// TIA Portal V20 export
FUNCTION_BLOCK "LAF_ManageAlarms"   // FB82, LAD
TITLE = LAF_ManageAlarms
AUTHOR : Siemens Digital Industries
FAMILY : LAF
// Mapping the ProDiag categories to the commands of the ModeStateManager.
// stored: Access Published, IsIECCheckEnabled true, MemoryReserve 100, SetENOAutomatically true
   VAR_INPUT
      proDiagState : SV_FB_State_V2;
   END_VAR
   VAR_OUTPUT
      parentAlarmDB : "LAF_typeAlarms";
      alarmDB : "LAF_typeAlarms";
      hmiInterfaceDB : "LAF_typeAlarms";
   END_VAR
   VAR_IN_OUT
      feedback : "LUC_typeEmFeedback";
   END_VAR
   VAR_TEMP
      temp : Bool;
   END_VAR
   VAR CONSTANT
      REPLACE : Bool;   // OEM: replace with ProDiag statuses that command unit state
   END_VAR
BEGIN

REGION Network 1: BLOCK INFO HEADER
   // SIEMENS AG / (c)Copyright 2024
   // ------------------------------------------------------------------------------
   // Title:            LAF_ManageAlarms
   // Comment/Function: Mapping the ProDiag categories to the commands of the ModeStateManager.
   // Library/Family:   Library of Automation Framework
   // Author:           Siemens Digital Industry
   // Tested with:      ---
   // Engineering:      TIA Portal V19
   // Restrictions:     -
   // Requirements:     ---
   // ------------------------------------------------------------------------------
   // Change log table:
   // Version  | Date       | Expert in charge       | Changes applied
   // ---------|------------|------------------------|------------------------------
   // 01.01.00 | 21.06.2024 | SIMATIC Systems Support
   //                         First released version
END_REGION

REGION Network 2: Stop command
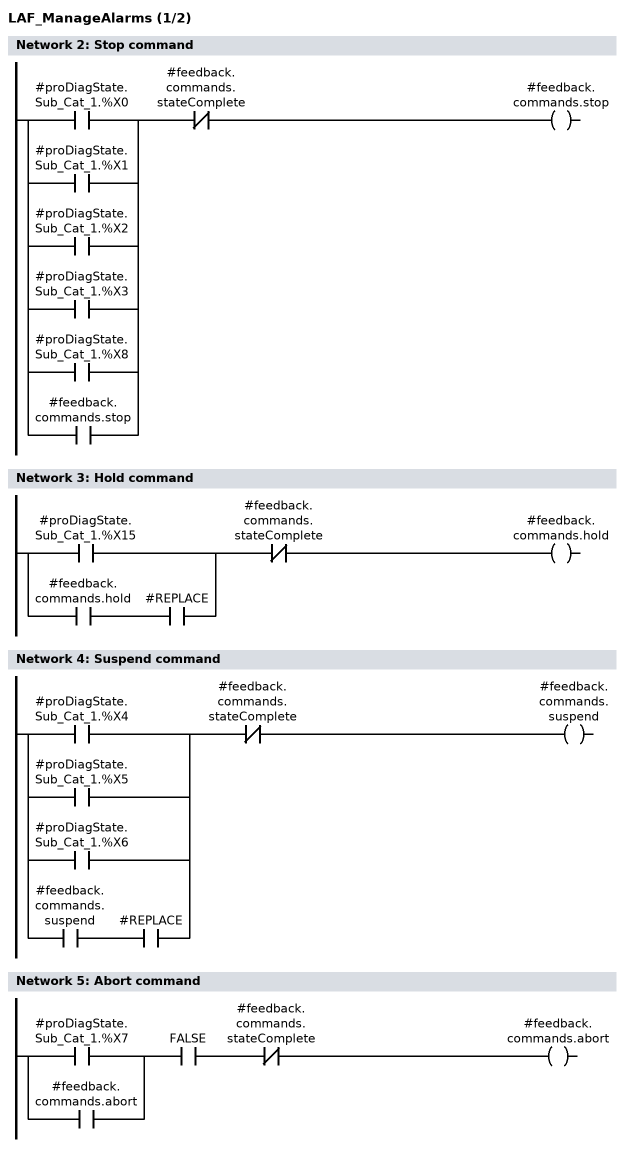
   RUNG wire#powerrail
      Contact( #proDiagState.Sub_Cat_1.%X0 )
      wire#w1
      I_Contact( #feedback.commands.stateComplete )
      Coil( #feedback.commands.stop )
   END_RUNG
   RUNG wire#powerrail
      Contact( #proDiagState.Sub_Cat_1.%X1 )
   END_RUNG wire#w1
   RUNG wire#powerrail
      Contact( #proDiagState.Sub_Cat_1.%X2 )
   END_RUNG wire#w1
   RUNG wire#powerrail
      Contact( #proDiagState.Sub_Cat_1.%X3 )
   END_RUNG wire#w1
   RUNG wire#powerrail
      Contact( #proDiagState.Sub_Cat_1.%X8 )
   END_RUNG wire#w1
   RUNG wire#powerrail
      Contact( #feedback.commands.stop )
   END_RUNG wire#w1
   // the same network as SCL:
   #feedback.commands.stop := (#proDiagState.Sub_Cat_1.%X0 OR #proDiagState.Sub_Cat_1.%X1 OR #proDiagState.Sub_Cat_1.%X2 OR #proDiagState.Sub_Cat_1.%X3 OR #proDiagState.Sub_Cat_1.%X8 OR #feedback.commands.stop) AND NOT #feedback.commands.stateComplete;
END_REGION

REGION Network 3: Hold command
   RUNG wire#powerrail
      Contact( #proDiagState.Sub_Cat_1.%X15 )
      wire#w1
      I_Contact( #feedback.commands.stateComplete )
      Coil( #feedback.commands.hold )
   END_RUNG
   RUNG wire#powerrail
      Contact( #feedback.commands.hold )
      Contact( #REPLACE )
   END_RUNG wire#w1
   // the same network as SCL:
   #feedback.commands.hold := (#proDiagState.Sub_Cat_1.%X15 OR (#feedback.commands.hold AND #REPLACE)) AND NOT #feedback.commands.stateComplete;
END_REGION

REGION Network 4: Suspend command
   RUNG wire#powerrail
      Contact( #proDiagState.Sub_Cat_1.%X4 )
      wire#w1
      I_Contact( #feedback.commands.stateComplete )
      Coil( #feedback.commands.suspend )
   END_RUNG
   RUNG wire#powerrail
      Contact( #proDiagState.Sub_Cat_1.%X5 )
   END_RUNG wire#w1
   RUNG wire#powerrail
      Contact( #proDiagState.Sub_Cat_1.%X6 )
   END_RUNG wire#w1
   RUNG wire#powerrail
      Contact( #feedback.commands.suspend )
      Contact( #REPLACE )
   END_RUNG wire#w1
   // the same network as SCL:
   #feedback.commands.suspend := (#proDiagState.Sub_Cat_1.%X4 OR #proDiagState.Sub_Cat_1.%X5 OR #proDiagState.Sub_Cat_1.%X6 OR (#feedback.commands.suspend AND #REPLACE)) AND NOT #feedback.commands.stateComplete;
END_REGION

REGION Network 5: Abort command
   RUNG wire#powerrail
      Contact( #proDiagState.Sub_Cat_1.%X7 )
      wire#w1
      Contact( FALSE )
      I_Contact( #feedback.commands.stateComplete )
      Coil( #feedback.commands.abort )
   END_RUNG
   RUNG wire#powerrail
      Contact( #feedback.commands.abort )
   END_RUNG wire#w1
   // the same network as SCL:
   #feedback.commands.abort := (#proDiagState.Sub_Cat_1.%X7 OR #feedback.commands.abort) AND FALSE AND NOT #feedback.commands.stateComplete;
END_REGION

REGION Network 6: Error State
   // MF, PF, TFIB, TFS, and SF are errors
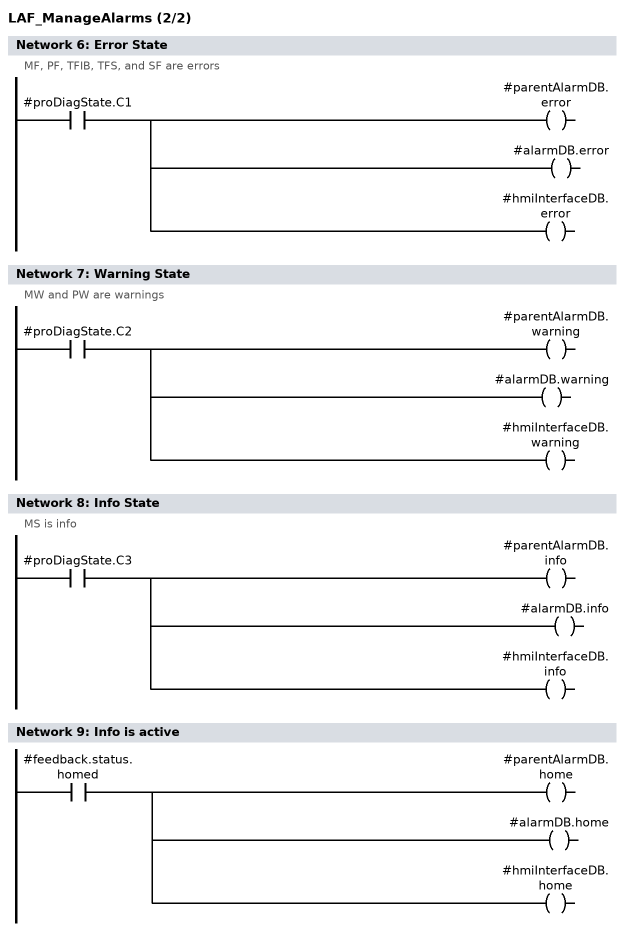
   RUNG wire#powerrail
      Contact( #proDiagState.C1 )
      wire#w1
      Coil( #parentAlarmDB.error )
   END_RUNG
   RUNG wire#w1
      Coil( #alarmDB.error )
   END_RUNG
   RUNG wire#w1
      Coil( #hmiInterfaceDB.error )
   END_RUNG
   // the same network as SCL:
   #parentAlarmDB.error := #proDiagState.C1;
   #alarmDB.error := #proDiagState.C1;
   #hmiInterfaceDB.error := #proDiagState.C1;
END_REGION

REGION Network 7: Warning State
   // MW and PW are warnings
   RUNG wire#powerrail
      Contact( #proDiagState.C2 )
      wire#w1
      Coil( #parentAlarmDB.warning )
   END_RUNG
   RUNG wire#w1
      Coil( #alarmDB.warning )
   END_RUNG
   RUNG wire#w1
      Coil( #hmiInterfaceDB.warning )
   END_RUNG
   // the same network as SCL:
   #parentAlarmDB.warning := #proDiagState.C2;
   #alarmDB.warning := #proDiagState.C2;
   #hmiInterfaceDB.warning := #proDiagState.C2;
END_REGION

REGION Network 8: Info State
   // MS is info
   RUNG wire#powerrail
      Contact( #proDiagState.C3 )
      wire#w1
      Coil( #parentAlarmDB.info )
   END_RUNG
   RUNG wire#w1
      Coil( #alarmDB.info )
   END_RUNG
   RUNG wire#w1
      Coil( #hmiInterfaceDB.info )
   END_RUNG
   // the same network as SCL:
   #parentAlarmDB.info := #proDiagState.C3;
   #alarmDB.info := #proDiagState.C3;
   #hmiInterfaceDB.info := #proDiagState.C3;
END_REGION

REGION Network 9: Info is active
   RUNG wire#powerrail
      Contact( #feedback.status.homed )
      wire#w1
      Coil( #parentAlarmDB.home )
   END_RUNG
   RUNG wire#w1
      Coil( #alarmDB.home )
   END_RUNG
   RUNG wire#w1
      Coil( #hmiInterfaceDB.home )
   END_RUNG
   // the same network as SCL:
   #parentAlarmDB.home := #feedback.status.homed;
   #alarmDB.home := #feedback.status.homed;
   #hmiInterfaceDB.home := #feedback.status.homed;
END_REGION
END_FUNCTION_BLOCK
